Staubli VAL3: stop.pgx

program stop()
begin

  //test command

end
